// TIA Portal project "ProjektPlcSimAdvTest" (V16)

(* hardware
DEVICE "S71500/ET200MP-Station_1"  S7-1500 station
   slot 0: "Profilschiene_0"  Rack  6ES7 590-1***0-0AA0
   slot 1: "PLC_1"  CPU 1515F-2 PN  6ES7 515-2FM02-0AB0  V2.8
      slot 3: "CPU-Display_1"  6ES7591-1BA00-0AA0
      slot 32768: "PROFINET-Schnittstelle_1"  X1
         slot 32769: "Port_1"  X1 P1
         slot 32770: "Port_2"  X1 P2
      slot 33024: "PROFINET-Schnittstelle_2"  X2
         slot 33025: "Port_1"  X2 P1
      slot 34817: "Virtual CP interface port_1"  Virtual CP interface port  Virtual CP interface port
*)

// ===== PLC "PLC_1"  CPU 1515F-2 PN =====

VAR_GLOBAL   // PLC tag table "Standard-Variablentabelle"
   "Eingang_01" AT %I0.0 : Bool;
   "Eingang_02" AT %I0.1 : Bool;
   "Eingang_03" AT %I0.2 : Bool;
   "Eingang_04" AT %I0.3 : Bool;
   "Eingang_05" AT %I0.4 : Bool;
   "Eingang_06" AT %I0.5 : Bool;
   "Eingang_07" AT %I0.6 : Bool;
   "Eingang_08" AT %I0.7 : Bool;
   "Ausgang_01" AT %Q1.0 : Bool;
   "Ausgang_02" AT %Q1.1 : Bool;
   "Ausgang_03" AT %Q1.2 : Bool;
   "Ausgang_04" AT %Q1.3 : Bool;
   "Ausgang_05" AT %Q1.4 : Bool;
   "Ausgang_06" AT %Q1.5 : Bool;
   "Ausgang_07" AT %Q1.6 : Bool;
   "Ausgang_08" AT %Q1.7 : Bool;
   "System_Byte" AT %MB1 : Byte;
   "FirstScan" AT %M1.0 : Bool;
   "DiagStatusUpdate" AT %M1.1 : Bool;
   "AlwaysTRUE" AT %M1.2 : Bool;
   "AlwaysFALSE" AT %M1.3 : Bool;
   "Clock_Byte" AT %MB10 : Byte;
   "Clock_10Hz" AT %M10.0 : Bool;
   "Clock_5Hz" AT %M10.1 : Bool;
   "Clock_2.5Hz" AT %M10.2 : Bool;
   "Clock_2Hz" AT %M10.3 : Bool;
   "Clock_1.25Hz" AT %M10.4 : Bool;
   "Clock_1Hz" AT %M10.5 : Bool;
   "Clock_0.625Hz" AT %M10.6 : Bool;
   "Clock_0.5Hz" AT %M10.7 : Bool;
   "Value_Set" AT %MW20 : Int;
   "Value_Actual" AT %MW22 : Int;
   "Value_Target" AT %MW24 : Int;
   "Set_Value" AT %M28.0 : Bool;
   "Start_Value" AT %M28.1 : Bool;
   "Value_Gradient" AT %MW26 : Int;
END_VAR

DATA_BLOCK "Main_Safety_RTG1_DB"   // DB1, F_DB
{ S7_Optimized_Access := 'TRUE' }
NAME : FUSI
VERSION : 0.1
// stored: InstanceOfName Main_Safety_RTG1
"Main_Safety_RTG1"
BEGIN
END_DATA_BLOCK

FUNCTION_BLOCK "Main_Safety_RTG1"   // FB1, F_FBD
{ S7_Optimized_Access := 'TRUE' }
BEGIN
END_FUNCTION_BLOCK

ORGANIZATION_BLOCK "Main"   // OB1, LAD, ProgramCycle
TITLE = "Main Program Sweep (Cycle)"
{ S7_Optimized_Access := 'TRUE' }
VERSION : 0.1
   VAR_INPUT
      Initial_Call : Bool;   // Initial call of this OB
      Remanence : Bool;   // =True, if remanent data are available
   END_VAR
BEGIN

REGION Network 1
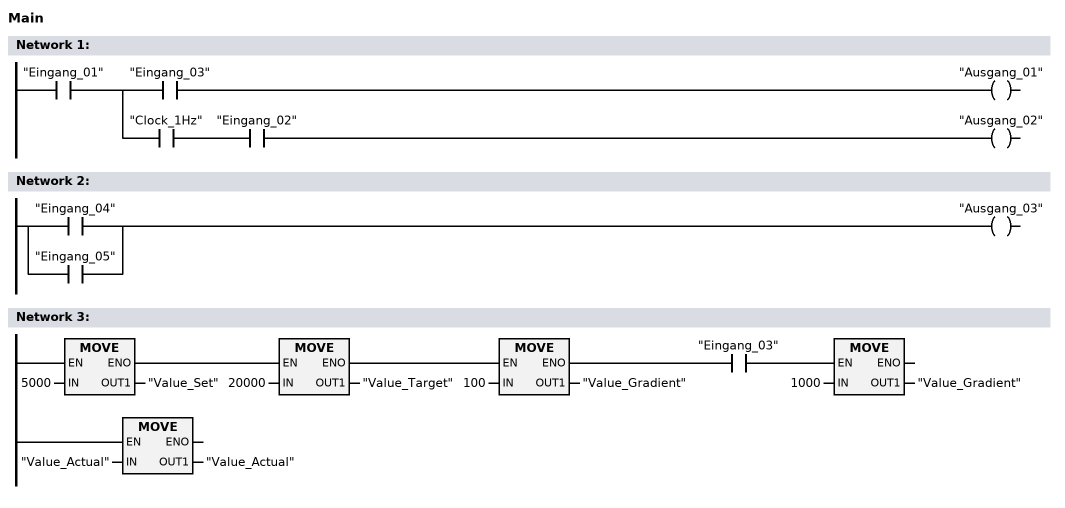
   RUNG wire#powerrail
      Contact( "Eingang_01" )
      wire#w1
      Contact( "Eingang_03" )
      Coil( "Ausgang_01" )
   END_RUNG
   RUNG wire#w1
      Contact( "Clock_1Hz" )
      Contact( "Eingang_02" )
      Coil( "Ausgang_02" )
   END_RUNG
   // the same network as SCL:
   "Ausgang_01" := "Eingang_01" AND "Eingang_03";
   "Ausgang_02" := "Eingang_01" AND "Clock_1Hz" AND "Eingang_02";
END_REGION

REGION Network 2
   RUNG wire#powerrail
      Contact( "Eingang_04" )
      wire#w1
      Coil( "Ausgang_03" )
   END_RUNG
   RUNG wire#powerrail
      Contact( "Eingang_05" )
   END_RUNG wire#w1
   // the same network as SCL:
   "Ausgang_03" := "Eingang_04" OR "Eingang_05";
END_REGION

REGION Network 3
   RUNG wire#powerrail
      Move(in := 5000, out1 => "Value_Set")
      Move(in := 20000, out1 => "Value_Target")
      Move(in := 100, out1 => "Value_Gradient")
      Contact( "Eingang_03" )
      Move(in := 1000, out1 => "Value_Gradient")
   END_RUNG
   RUNG wire#powerrail
      Move(in := "Value_Actual", out1 => "Value_Actual")
   END_RUNG
   // the same network as SCL:
   "Value_Set" := 5000;
   "Value_Target" := 20000;
   "Value_Gradient" := 100;
   IF "Eingang_03" THEN "Value_Gradient" := 1000; END_IF;
   "Value_Actual" := "Value_Actual";
END_REGION
END_ORGANIZATION_BLOCK